RoboDK station: Example 3 - Unload pallet - Start.rdk

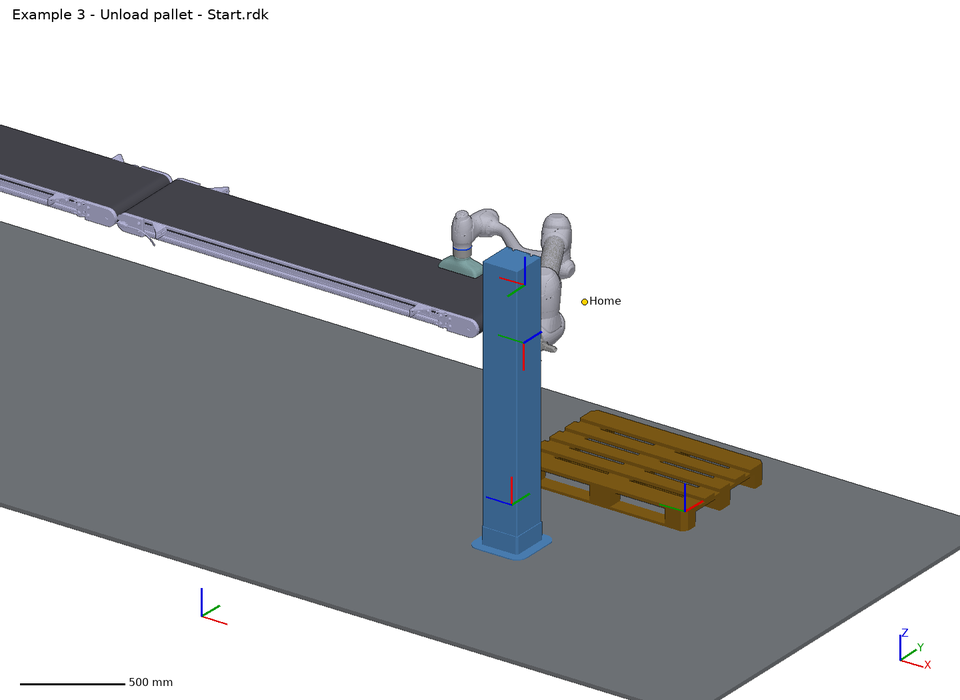
[picture v0: the station drawn from its stored meshes, robots at their saved joint values, targets as dots, program paths as lines]
Station Example 3 - Unload pallet. Poses are relative to the parent item; angles as X-Y-Z fixed-axis rotations.
  - frame Linear Rail Base at (750, 1500, 200) mm, rotated rx 0 ry -90 rz 0 deg
    - robot Linear Rail: 1 axes
        modified DH rows (alpha deg, a mm, theta deg, d mm): 0, 0, 0, 0 linear
        base shift (0, 0, 0) mm, rotated rx 0 ry 90 rz 0 deg
        joint limits [0] to [1200]; home [0]; saved at [819.16]
      - frame Doosan Robotics M1013 Base at (0, 100, 0) mm, rotated rx 90 ry 0 rz 180 deg
        - robot Doosan Robotics M1013: 6 axes, payload 10 kg, reach 1300 mm, repeatability 0.1 mm, weight 33 kg
            modified DH rows (alpha deg, a mm, theta deg, d mm): 0, 0, 0, 152.5; -90, 0, -90, 34.506; 0, 620, -90, 0; -90, 0, 0, 559; 90, 0, 0, 0; -90, 0, 180, 121
            base shift (0, 0, 0) mm, rotated rx 0 ry 0 rz 180 deg
            joint limits [-120, -100, -160, -360, -360, -360] to [-60, 100, 160, 360, 360, 360]; home [0, 0, -90, 0, 0, 0]; saved at [-88.76, 29.09, 58.79, 89.94, -91.21, -92.1]
          - tool Tool, TCP at (0, 0, 69) mm, size 225 x 100 x 69 mm, geometry from Tool.step
  - frame Conveyor Belt Base at (57.17, 2600, 730) mm, rotated rx 0 ry 0 rz -180 deg
    - robot Conveyor Belt: 1 axes
        modified DH rows (alpha deg, a mm, theta deg, d mm): 0, 0, 0, 0 linear
        base shift (0, 0, 0) mm, rotated rx 0 ry 90 rz 0 deg
        joint limits [-500000] to [500000]; home [0]; saved at [-494045.004]
      - frame Conveyor at (0, 0, 0) mm
    - object Conveyor at (2400, 440, -50) mm, rotated rx 0 ry 0 rz -90 deg, size 597 x 2090.8 x 107.2 mm
    - object Conveyor at (4500, 440, -50) mm, rotated rx 0 ry 0 rz -90 deg, size 597 x 2090.8 x 107.2 mm
  - frame Pallet at (1350, 2080, 100) mm, rotated rx 0 ry 0 rz 90 deg
    - object Pallet at (-0.19, 0.17, 1.21) mm, size 660 x 990 x 118.8 mm, geometry from User Library-Europallet.igs
  - frame World at (0, 0, 0) mm
    - target Home (joint target) at (876.47, 1924.34, 1140.31) mm, rotated rx -180 ry 0 rz 0 deg; joints [-90, -100, 160, 90, -90, -120, 1095.8] of Doosan Robotics M1013
    - target ConvHome (Cartesian target) at (500057.17, 2600, 730) mm, rotated rx 0 ry 0 rz -180 deg; joints [-500000, 0, 0, 0, 0, 0, 0] of Conveyor Belt
    - target ConvRun (Cartesian target) at (392.51, 2433.37, 999.75) mm, rotated rx 180 ry 0 rz 2.38 deg; joints [50000, -58.983, -101.068, -19.936, -5.281, -2.394, 1150.26] of Conveyor Belt
    - object Floor at (-7500, 480, -30) mm, size 10000 x 2500 x 20 mm, geometry from Floor.step
  - program ReplaceObjects (1 instructions, listed below)
  - program MainProgram (0 instructions, listed below)
  - program AppPallet (0 instructions, listed below)
  - program DropConveyor (0 instructions, listed below)
  - program GoHome (0 instructions, listed below)
  - program Pick (0 instructions, listed below)
  - program RunConveyor (2 instructions, listed below)

--- program ReplaceObjects (robot Doosan Robotics M1013) ---
  Replace objects

--- program MainProgram ---

--- program AppPallet ---

--- program DropConveyor ---

--- program GoHome ---

--- program Pick ---

--- program RunConveyor (robot Conveyor Belt) ---
  Set Ref.: World
  MoveJ (ConvRun)
